Omron CX-Programmer project PampaBlanca (CX-Programmer 7.21)

# PLC PLC: CJ1M CPU13
I/O table (CPU CJ1M-CPU13): rack 0 slot 0 CJ1W-ETN21(ETN11Mode); rack 0 slot 1 CJ1W-SRM21(2CH); rack 0 slot 2 CJ1W-ID261; rack 0 slot 3 CJ1W-ID261; rack 0 slot 4 CJ1W-ID261; rack 0 slot 5 CJ1W-OD261; rack 0 slot 6 CJ1W-OD261; rack 0 slot 7 CJ1W-OD231

## Global symbols (name address type ; comment)
AFRE 2000.03 BOOL L
BLZ1 2001.06 BOOL L
BLZ2 12.02 BOOL L
BLZ4 12.03 BOOL L
BLZ5 12.04 BOOL L
BLZ6 12.05 BOOL L
EMERGENCIA W300.00 BOOL L
EVM32 2001.07 BOOL L
EVM48 2001.08 BOOL L
EVM5 2001.04 BOOL L
EVMN25 2001.05 BOOL L
EVS11 2000.04 BOOL L
EVS11_C 2000.05 BOOL L
EVS12 2000.06 BOOL L
EVS12_C 2000.07 BOOL L
EVS13P 2000.08 BOOL L
EVS13P_C 2000.09 BOOL L
EVS13S 2000.10 BOOL L
EVS13S_C 2000.11 BOOL L
HAR2 2000.00 BOOL L
HARI 2000.02 BOOL L
M1 20.00 BOOL L
M10 20.12 BOOL L
M100 19.13 BOOL L
M102 19.14 BOOL L
M103 19.15 BOOL L
M104 2002.01 BOOL L
M105 14.00 BOOL L
M106 14.01 BOOL L
M107 14.02 BOOL L
M108 14.03 BOOL L
M108A 14.04 BOOL L
M11 20.13 BOOL L
M116 14.05 BOOL L
M117 14.06 BOOL L
M117A 14.07 BOOL L
M118 14.08 BOOL L
M11A 20.14 BOOL L
M12 20.15 BOOL L
M13 21.00 BOOL L
M14 21.01 BOOL L
M15 21.02 BOOL L
M152 12.07 BOOL L
M153 14.09 BOOL L  ; BALANZA AFRECHO CONTACTOR  C93
M153Z 12.08 BOOL L
M16 21.03 BOOL L
M16A 21.04 BOOL L
M17 21.05 BOOL L
M2 20.01 BOOL L
M21 21.06 BOOL L
M22 21.07 BOOL L
M23 21.08 BOOL L
M3 20.02 BOOL L
M31 21.09 BOOL L
M32 21.10 BOOL L
M34 21.11 BOOL L
M35 21.12 BOOL L
M36 21.13 BOOL L
M37 21.14 BOOL L
M37A 21.15 BOOL L
M38 18.00 BOOL L
M3A 20.03 BOOL L
M3B 20.04 BOOL L
M4 20.05 BOOL L
M46 18.01 BOOL L
M47 18.02 BOOL L
M48 18.03 BOOL L
M5 20.06 BOOL L
M50 18.04 BOOL L
M50A 18.05 BOOL L
M51 18.06 BOOL L
M51A 18.07 BOOL L
M52 18.08 BOOL L
M53 18.09 BOOL L
M54 18.10 BOOL L
M55 18.11 BOOL L
M56 18.12 BOOL L
M58 18.13 BOOL L
M59 18.14 BOOL L
M6 20.07 BOOL L
M61 18.15 BOOL L
M62 19.00 BOOL L
M63 19.01 BOOL L
M64 19.02 BOOL L
M65 19.03 BOOL L
M69 19.04 BOOL L
M7 20.08 BOOL L
M70 19.05 BOOL L
M71 19.06 BOOL L
M73 19.07 BOOL L
M75 19.08 BOOL L
M7A 20.09 BOOL L
M8 20.10 BOOL L
M9 20.11 BOOL L
M91 2002.00 BOOL L
M95 19.09 BOOL L
M96 19.10 BOOL L
M97 19.11 BOOL L
M99 19.12 BOOL L
MI 2002.02 BOOL L
MII 2002.03 BOOL L
MN1 14.11 BOOL L
MN10 2002.06 BOOL L
MN100 2002.10 BOOL L
MN11 14.15 BOOL L
MN12 15.00 BOOL L
MN13 2002.07 BOOL L
MN14 2002.08 BOOL L
MN15 2002.09 BOOL L
MN16 15.01 BOOL L
MN17 15.02 BOOL L
MN18 15.03 BOOL L
MN2 14.12 BOOL L
MN21 15.04 BOOL L
MN24 15.05 BOOL L
MN25 15.06 BOOL L
MN26 15.07 BOOL L
MN27 15.08 BOOL L
MN28 15.09 BOOL L
MN3 14.13 BOOL L
MN35 15.12 BOOL L
MN36 15.11 BOOL L
MN37 15.10 BOOL L
MN4 14.14 BOOL L
MN9 2002.05 BOOL L
MOZD 2000.01 BOOL L
MV 2002.04 BOOL L
MVIII 14.10 BOOL L
MYFA 12.06 BOOL L
R1MN24 2001.02 BOOL L
R1MN24_C 2001.03 BOOL L
R1MN26 2001.00 BOOL L
R1MN26_C 2001.01 BOOL L
R2MN24 2002.11 BOOL L
R2MN24_C 2002.12 BOOL L
R2MN26 2000.14 BOOL L
R2MN26_C 2000.15 BOOL L
R3MN26 2000.12 BOOL L
R3MN26_C 2000.13 BOOL L
RST32 15.14 BOOL L
RST48 15.15 BOOL L
STOP W300.01 BOOL L
TBEHA 15.13 BOOL L  ; EMBOLSADO HARIN CONTACTOR C92
XBT13 2012.15 BOOL L
XEMER0 7.11 BOOL L
XEMER1 7.10 BOOL L
XFCCM32 2008.13 BOOL L
XFCCM48 2011.10 BOOL L
XFCMN24 2008.08 BOOL L
XFCMN26 2008.09 BOOL L
XFCMN37 7.04 BOOL L
XFCMVIII 2008.10 BOOL L
XFCOM32 2008.12 BOOL L
XFCOM48 2011.09 BOOL L
XHABI1 7.09 BOOL L
XM1 0.00 BOOL L
XM10 0.12 BOOL L
XM100 4.00 BOOL L
XM102 4.01 BOOL L
XM103 4.02 BOOL L
XM104 2012.14 BOOL L
XM105 4.03 BOOL L
XM106 4.04 BOOL L
XM107 4.05 BOOL L
XM108 4.06 BOOL L
XM108A 4.07 BOOL L
XM11 0.13 BOOL L
XM116 4.08 BOOL L
XM117 4.09 BOOL L
XM117A 4.10 BOOL L
XM118 4.11 BOOL L
XM11A 0.14 BOOL L
XM12 0.15 BOOL L
XM13 1.00 BOOL L
XM14 1.01 BOOL L
XM15 1.02 BOOL L
XM153 4.12 BOOL L
XM16 1.03 BOOL L
XM16A 1.04 BOOL L
XM17 1.05 BOOL L
XM2 0.01 BOOL L
XM20 1.06 BOOL L
XM21 1.07 BOOL L
XM22 1.08 BOOL L
XM23 1.09 BOOL L
XM3 0.02 BOOL L
XM31 1.10 BOOL L
XM32 1.11 BOOL L
XM34 1.12 BOOL L
XM35 1.13 BOOL L
XM36 1.14 BOOL L
XM37 1.15 BOOL L
XM37A 2.00 BOOL L
XM38 2.01 BOOL L
XM3A 0.03 BOOL L
XM3B 0.04 BOOL L
XM4 0.05 BOOL L
XM46 2.02 BOOL L
XM47 2.03 BOOL L
XM48 2.04 BOOL L
XM5 0.06 BOOL L
XM50 2.05 BOOL L
XM50A 2.06 BOOL L
XM51 2.07 BOOL L
XM51A 2.08 BOOL L
XM52 2.09 BOOL L
XM53 2.10 BOOL L
XM54 2.11 BOOL L
XM55 2.12 BOOL L
XM56 2.13 BOOL L
XM58 2.14 BOOL L
XM59 2.15 BOOL L
XM6 0.07 BOOL L
XM61 3.00 BOOL L
XM62 3.01 BOOL L
XM63 3.02 BOOL L
XM64 3.03 BOOL L
XM65 3.04 BOOL L
XM69 3.05 BOOL L
XM7 0.08 BOOL L
XM70 3.06 BOOL L
XM71 3.07 BOOL L
XM73 3.08 BOOL L
XM75 3.09 BOOL L
XM7A 0.09 BOOL L
XM8 0.10 BOOL L
XM9 0.11 BOOL L
XM91 2012.12 BOOL L
XM92 3.10 BOOL L
XM93 3.11 BOOL L
XM95 3.12 BOOL L
XM96 3.13 BOOL L
XM97 3.14 BOOL L
XM99 3.15 BOOL L
XMI 2012.05 BOOL L
XMII 2012.06 BOOL L
XMN1 4.14 BOOL L
XMN10 2012.08 BOOL L
XMN100 2012.13 BOOL L
XMN11 5.02 BOOL L
XMN12 5.03 BOOL L
XMN13 2012.09 BOOL L
XMN14 2012.10 BOOL L
XMN15 2012.11 BOOL L
XMN16 5.04 BOOL L
XMN17 5.05 BOOL L
XMN18 5.06 BOOL L
XMN2 4.15 BOOL L
XMN21 5.07 BOOL L
XMN24 5.08 BOOL L
XMN25 5.09 BOOL L
XMN26 5.10 BOOL L
XMN27 5.11 BOOL L
XMN28 5.12 BOOL L
XMN3 5.00 BOOL L
XMN35 5.13 BOOL L
XMN36 5.14 BOOL L
XMN37 5.15 BOOL L
XMN4 5.01 BOOL L
XMN9 2012.07 BOOL L
XMVIII 4.13 BOOL L
XSAS1 2011.00 BOOL L
XSAS10 2011.08 BOOL L
XSAS11 2009.00 BOOL L
XSAS12 2009.05 BOOL L
XSAS13 2009.10 BOOL L
XSAS14 2008.14 BOOL L
XSAS15 2008.15 BOOL L
XSAS2 2011.01 BOOL L
XSAS3 2011.02 BOOL L
XSAS4 2011.03 BOOL L
XSAS5 2011.04 BOOL L
XSAS6 2011.05 BOOL L
XSAS7 2008.07 BOOL L
XSAS8 2011.06 BOOL L
XSAS9 2011.07 BOOL L
XSBS11 6.07 BOOL L
XSBS12 6.08 BOOL L
XSBS13 6.09 BOOL L
XSC1M54 2010.08 BOOL L
XSC1M55 2010.10 BOOL L
XSC2M54 2010.09 BOOL L
XSC2M55 2010.11 BOOL L
XSHM5 2008.11 BOOL L
XSHMN25 2010.02 BOOL L
XSIBLZ1 2010.15 BOOL L
XSIBLZ2 6.01 BOOL L
XSIBLZ5 6.04 BOOL L
XSIBLZ6 6.06 BOOL L
XSIC1MN26 2009.14 BOOL L
XSIC1S13 2009.12 BOOL L
XSIC2MN26 2009.09 BOOL L
XSIC2S13 2010.00 BOOL L
XSIC3MN26 2009.04 BOOL L
XSICR1MN24 2010.14 BOOL L
XSICR2MN24 2012.04 BOOL L
XSICS11 2009.01 BOOL L
XSICS12 2009.07 BOOL L
XSIO1MN26 2009.13 BOOL L
XSIO1S13 2009.11 BOOL L
XSIO2MN26 2009.08 BOOL L
XSIO2S13 2009.15 BOOL L
XSIO3MN26 2009.03 BOOL L
XSIOR1MN24 2010.13 BOOL L
XSIOR2MN24 2012.03 BOOL L
XSIOS11 2009.02 BOOL L
XSIOS12 2009.06 BOOL L
XSNAMN16 7.00 BOOL L
XSNBMN16 7.01 BOOL L
XSR1M61 7.05 BOOL L
XSR2M61 7.06 BOOL L
XSRM10 6.11 BOOL L
XSRM100 6.15 BOOL L
XSRM100_A 2008.06 BOOL L
XSRM10_A 2008.02 BOOL L
XSRM11 2008.03 BOOL L
XSRM11A 6.13 BOOL L
XSRM11A_A 2008.04 BOOL L
XSRM12 6.12 BOOL L
XSRM35 7.02 BOOL L
XSRM62 2010.04 BOOL L
XSRM63 2010.05 BOOL L
XSRM64 2010.06 BOOL L
XSRM65 2010.07 BOOL L
XSRM9 6.10 BOOL L
XSRM99 6.14 BOOL L
XSRM99_A 2008.05 BOOL L
XSRM9_A 2008.01 BOOL L
XSRMN100 2012.02 BOOL L
XSRMN102 7.07 BOOL L
XSRMN103 7.08 BOOL L
XSRMN24 2010.12 BOOL L
XSRMN26 2010.03 BOOL L
XSRMN37 7.03 BOOL L
XSSBLZ1 2010.01 BOOL L
XSSBLZ2 6.00 BOOL L
XSSBLZ4 6.02 BOOL L
XSSBLZ5 6.03 BOOL L
XSSBLZ6 6.05 BOOL L
XSTMN14INF 2012.01 BOOL L
XSTMN14SUP 2012.00 BOOL L
YAFRE W499.03 BOOL L
YBLZ1 W498.06 BOOL L
YBLZ2 W506.02 BOOL L
YBLZ4 W506.03 BOOL L
YBLZ5 W506.04 BOOL L
YBLZ6 W506.05 BOOL L
YEVM32 W498.07 BOOL L
YEVM48 W498.08 BOOL L
YEVM5 W498.04 BOOL L
YEVMN25 W498.05 BOOL L
YEVS11 W499.04 BOOL L
YEVS11_C W499.05 BOOL L
YEVS12 W499.06 BOOL L
YEVS12_C W499.07 BOOL L
YEVS13P W499.08 BOOL L
YEVS13P_C W499.09 BOOL L
YEVS13S W499.10 BOOL L
YEVS13S_C W499.11 BOOL L
YHAR2 W499.00 BOOL L
YHARI W499.02 BOOL L
YM1 W500.00 BOOL L
YM10 W500.12 BOOL L
YM100 W503.13 BOOL L
YM102 W503.14 BOOL L
YM103 W503.15 BOOL L
YM104 W497.01 BOOL L
YM105 W504.00 BOOL L
YM106 W504.01 BOOL L
YM107 W504.02 BOOL L
YM108 W504.03 BOOL L
YM108A W504.04 BOOL L
YM11 W500.13 BOOL L
YM116 W504.05 BOOL L
YM117 W504.06 BOOL L
YM117A W504.07 BOOL L
YM118 W504.08 BOOL L
YM11A W500.14 BOOL L
YM12 W500.15 BOOL L
YM13 W501.00 BOOL L
YM14 W501.01 BOOL L
YM15 W501.02 BOOL L
YM152 W506.07 BOOL L
YM153 W504.09 BOOL L
YM153Z W506.08 BOOL L
YM16 W501.03 BOOL L
YM16A W501.04 BOOL L
YM17 W501.05 BOOL L
YM2 W500.01 BOOL L
YM21 W501.06 BOOL L
YM22 W501.07 BOOL L
YM23 W501.08 BOOL L
YM3 W500.02 BOOL L
YM31 W501.09 BOOL L
YM32 W501.10 BOOL L
YM34 W501.11 BOOL L
YM35 W501.12 BOOL L
YM36 W501.13 BOOL L
YM37 W501.14 BOOL L
YM37A W501.15 BOOL L
YM38 W502.00 BOOL L
YM3A W500.03 BOOL L
YM3B W500.04 BOOL L
YM4 W500.05 BOOL L
YM46 W502.01 BOOL L
YM47 W502.02 BOOL L
YM48 W502.03 BOOL L
YM5 W500.06 BOOL L
YM50 W502.04 BOOL L
YM50A W502.05 BOOL L
YM51 W502.06 BOOL L
YM51A W502.07 BOOL L
YM52 W502.08 BOOL L
YM53 W502.09 BOOL L
YM54 W502.10 BOOL L
YM55 W502.11 BOOL L
YM56 W502.12 BOOL L
YM58 W502.13 BOOL L
YM59 W502.14 BOOL L
YM6 W500.07 BOOL L
YM61 W502.15 BOOL L
YM62 W503.00 BOOL L
YM63 W503.01 BOOL L
YM64 W503.02 BOOL L
YM65 W503.03 BOOL L
YM69 W503.04 BOOL L
YM7 W500.08 BOOL L
YM70 W503.05 BOOL L
YM71 W503.06 BOOL L
YM73 W503.07 BOOL L
YM75 W503.08 BOOL L
YM7A W500.09 BOOL L
YM8 W500.10 BOOL L
YM9 W500.11 BOOL L
YM91 W497.00 BOOL L
YM95 W503.09 BOOL L
YM96 W503.10 BOOL L
YM97 W503.11 BOOL L
YM99 W503.12 BOOL L
YMI W497.02 BOOL L
YMII W497.03 BOOL L
YMN1 W504.11 BOOL L
YMN10 W497.06 BOOL L
YMN100 W497.10 BOOL L
YMN11 W504.15 BOOL L
YMN12 W505.00 BOOL L
YMN13 W497.07 BOOL L
YMN14 W497.08 BOOL L
YMN15 W497.09 BOOL L
YMN16 W505.01 BOOL L
YMN17 W505.02 BOOL L
YMN18 W505.03 BOOL L
YMN2 W504.12 BOOL L
YMN21 W505.04 BOOL L
YMN24 W505.05 BOOL L
YMN25 W505.06 BOOL L
YMN26 W505.07 BOOL L
YMN27 W505.08 BOOL L
YMN28 W505.09 BOOL L
YMN3 W504.13 BOOL L
YMN35 W505.12 BOOL L
YMN36 W505.11 BOOL L
YMN37 W505.10 BOOL L
YMN4 W504.14 BOOL L
YMN9 W497.05 BOOL L
YMOZD W499.01 BOOL L
YMV W497.04 BOOL L
YMVIII W504.10 BOOL L
YMYFA W506.06 BOOL L
YR1MN24 W498.02 BOOL L
YR1MN24_C W498.03 BOOL L
YR1MN26 W498.00 BOOL L
YR1MN26_C W498.01 BOOL L
YR2MN24 W497.11 BOOL L
YR2MN24_C W497.12 BOOL L
YR2MN26 W499.14 BOOL L
YR2MN26_C W499.15 BOOL L
YR3MN26 W499.12 BOOL L
YR3MN26_C W499.13 BOOL L
YRST32 W300.10 BOOL L
YRST48 W300.11 BOOL L
YTBEHA W505.13 BOOL L

## Program PRINCIPAL (cyclic task 0)
; MOLINO PAMPA BLANCA

### Section Emergencia

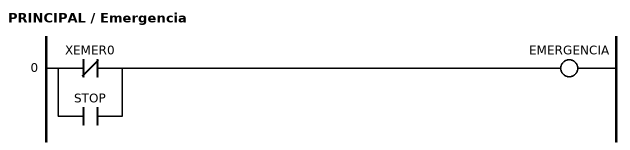
; rung 0
LDNOT XEMER0
OR STOP
OUT EMERGENCIA

### Section Llenar_Pellets_CTRL

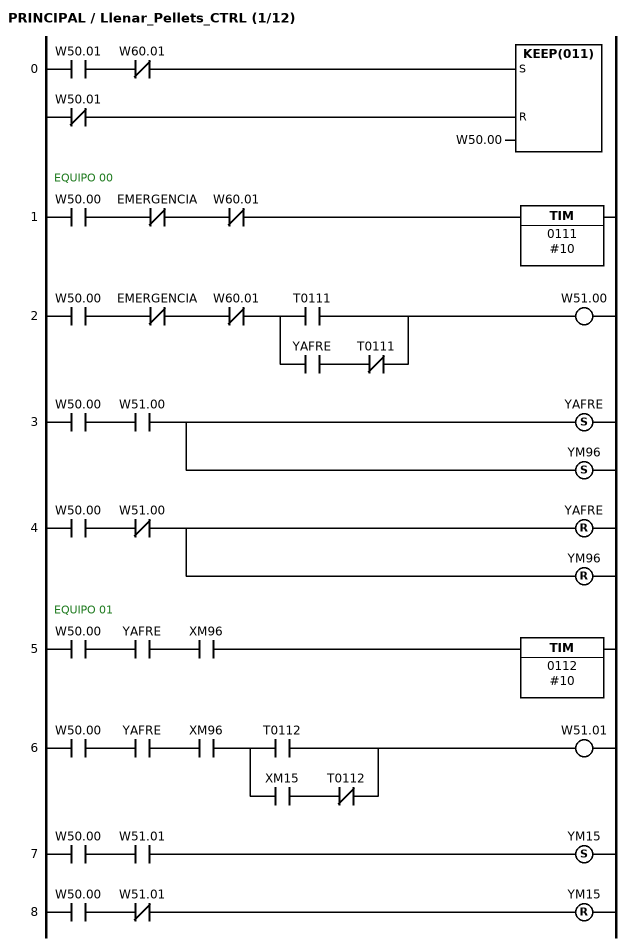
; rung 0
LD W50.01
ANDNOT W60.01
LDNOT W50.01
KEEP(011) W50.00
; rung 1: EQUIPO 00
LD W50.00
ANDNOT EMERGENCIA
ANDNOT W60.01
TIM 0111 #10
; rung 2
LD W50.00
ANDNOT EMERGENCIA
ANDNOT W60.01
LD T0111
LD YAFRE
ANDNOT T0111
ORLD
ANDLD
OUT W51.00
; rung 3
LD W50.00
AND W51.00
SET YAFRE
SET YM96
; rung 4
LD W50.00
ANDNOT W51.00
RSET YAFRE
RSET YM96
; rung 5: EQUIPO 01
LD W50.00
AND YAFRE
AND XM96
TIM 0112 #10
; rung 6
LD W50.00
AND YAFRE
AND XM96
LD T0112
LD XM15
ANDNOT T0112
ORLD
ANDLD
OUT W51.01
; rung 7
LD W50.00
AND W51.01
SET YM15
; rung 8
LD W50.00
ANDNOT W51.01
RSET YM15

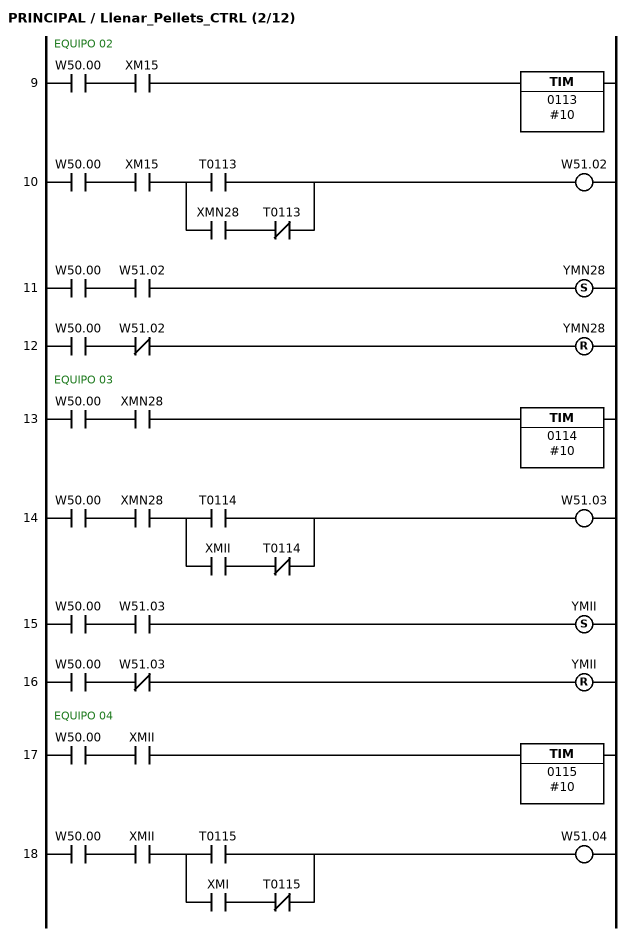
; rung 9: EQUIPO 02
LD W50.00
AND XM15
TIM 0113 #10
; rung 10
LD W50.00
AND XM15
LD T0113
LD XMN28
ANDNOT T0113
ORLD
ANDLD
OUT W51.02
; rung 11
LD W50.00
AND W51.02
SET YMN28
; rung 12
LD W50.00
ANDNOT W51.02
RSET YMN28
; rung 13: EQUIPO 03
LD W50.00
AND XMN28
TIM 0114 #10
; rung 14
LD W50.00
AND XMN28
LD T0114
LD XMII
ANDNOT T0114
ORLD
ANDLD
OUT W51.03
; rung 15
LD W50.00
AND W51.03
SET YMII
; rung 16
LD W50.00
ANDNOT W51.03
RSET YMII
; rung 17: EQUIPO 04
LD W50.00
AND XMII
TIM 0115 #10
; rung 18
LD W50.00
AND XMII
LD T0115
LD XMI
ANDNOT T0115
ORLD
ANDLD
OUT W51.04

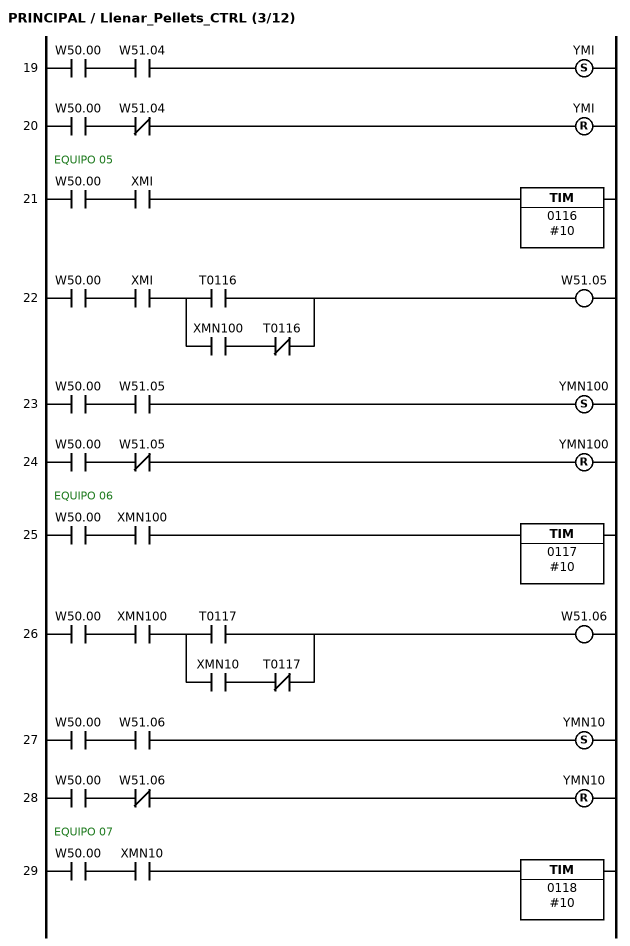
; rung 19
LD W50.00
AND W51.04
SET YMI
; rung 20
LD W50.00
ANDNOT W51.04
RSET YMI
; rung 21: EQUIPO 05
LD W50.00
AND XMI
TIM 0116 #10
; rung 22
LD W50.00
AND XMI
LD T0116
LD XMN100
ANDNOT T0116
ORLD
ANDLD
OUT W51.05
; rung 23
LD W50.00
AND W51.05
SET YMN100
; rung 24
LD W50.00
ANDNOT W51.05
RSET YMN100
; rung 25: EQUIPO 06
LD W50.00
AND XMN100
TIM 0117 #10
; rung 26
LD W50.00
AND XMN100
LD T0117
LD XMN10
ANDNOT T0117
ORLD
ANDLD
OUT W51.06
; rung 27
LD W50.00
AND W51.06
SET YMN10
; rung 28
LD W50.00
ANDNOT W51.06
RSET YMN10
; rung 29: EQUIPO 07
LD W50.00
AND XMN10
TIM 0118 #10

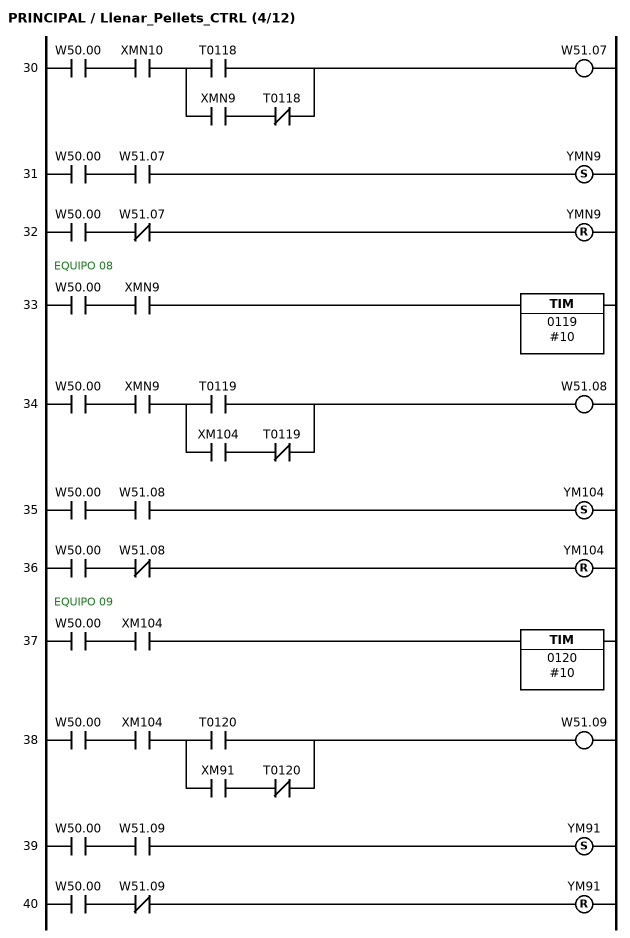
; rung 30
LD W50.00
AND XMN10
LD T0118
LD XMN9
ANDNOT T0118
ORLD
ANDLD
OUT W51.07
; rung 31
LD W50.00
AND W51.07
SET YMN9
; rung 32
LD W50.00
ANDNOT W51.07
RSET YMN9
; rung 33: EQUIPO 08
LD W50.00
AND XMN9
TIM 0119 #10
; rung 34
LD W50.00
AND XMN9
LD T0119
LD XM104
ANDNOT T0119
ORLD
ANDLD
OUT W51.08
; rung 35
LD W50.00
AND W51.08
SET YM104
; rung 36
LD W50.00
ANDNOT W51.08
RSET YM104
; rung 37: EQUIPO 09
LD W50.00
AND XM104
TIM 0120 #10
; rung 38
LD W50.00
AND XM104
LD T0120
LD XM91
ANDNOT T0120
ORLD
ANDLD
OUT W51.09
; rung 39
LD W50.00
AND W51.09
SET YM91
; rung 40
LD W50.00
ANDNOT W51.09
RSET YM91

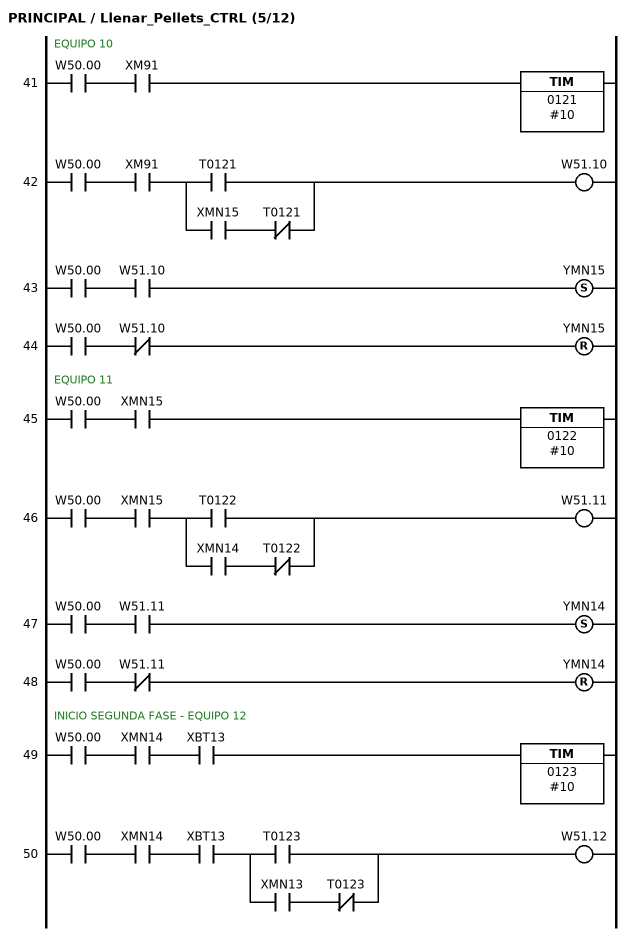
; rung 41: EQUIPO 10
LD W50.00
AND XM91
TIM 0121 #10
; rung 42
LD W50.00
AND XM91
LD T0121
LD XMN15
ANDNOT T0121
ORLD
ANDLD
OUT W51.10
; rung 43
LD W50.00
AND W51.10
SET YMN15
; rung 44
LD W50.00
ANDNOT W51.10
RSET YMN15
; rung 45: EQUIPO 11
LD W50.00
AND XMN15
TIM 0122 #10
; rung 46
LD W50.00
AND XMN15
LD T0122
LD XMN14
ANDNOT T0122
ORLD
ANDLD
OUT W51.11
; rung 47
LD W50.00
AND W51.11
SET YMN14
; rung 48
LD W50.00
ANDNOT W51.11
RSET YMN14
; rung 49: INICIO SEGUNDA FASE - EQUIPO 12
LD W50.00
AND XMN14
AND XBT13
TIM 0123 #10
; rung 50
LD W50.00
AND XMN14
AND XBT13
LD T0123
LD XMN13
ANDNOT T0123
ORLD
ANDLD
OUT W51.12

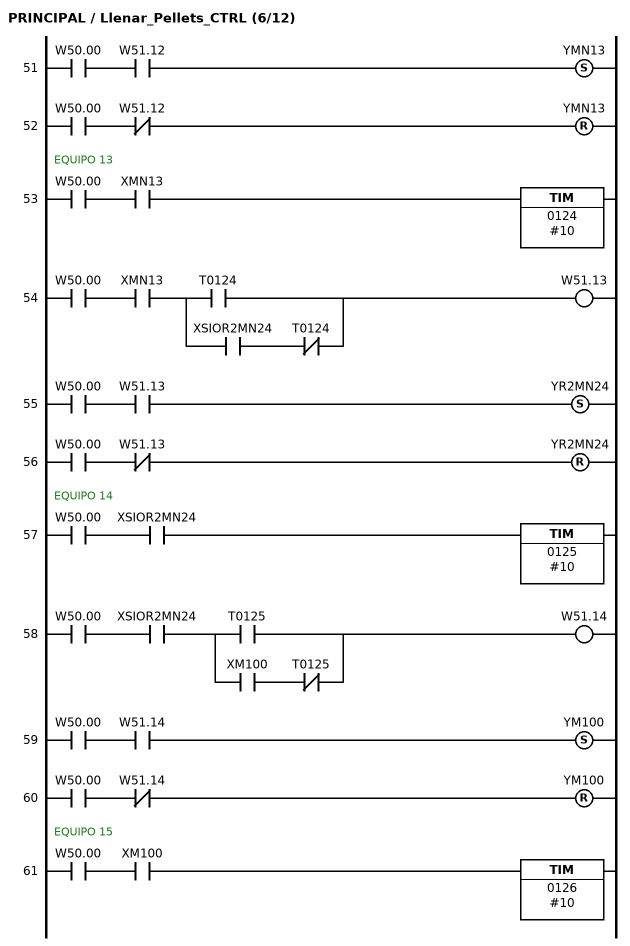
; rung 51
LD W50.00
AND W51.12
SET YMN13
; rung 52
LD W50.00
ANDNOT W51.12
RSET YMN13
; rung 53: EQUIPO 13
LD W50.00
AND XMN13
TIM 0124 #10
; rung 54
LD W50.00
AND XMN13
LD T0124
LD XSIOR2MN24
ANDNOT T0124
ORLD
ANDLD
OUT W51.13
; rung 55
LD W50.00
AND W51.13
SET YR2MN24
; rung 56
LD W50.00
ANDNOT W51.13
RSET YR2MN24
; rung 57: EQUIPO 14
LD W50.00
AND XSIOR2MN24
TIM 0125 #10
; rung 58
LD W50.00
AND XSIOR2MN24
LD T0125
LD XM100
ANDNOT T0125
ORLD
ANDLD
OUT W51.14
; rung 59
LD W50.00
AND W51.14
SET YM100
; rung 60
LD W50.00
ANDNOT W51.14
RSET YM100
; rung 61: EQUIPO 15
LD W50.00
AND XM100
TIM 0126 #10

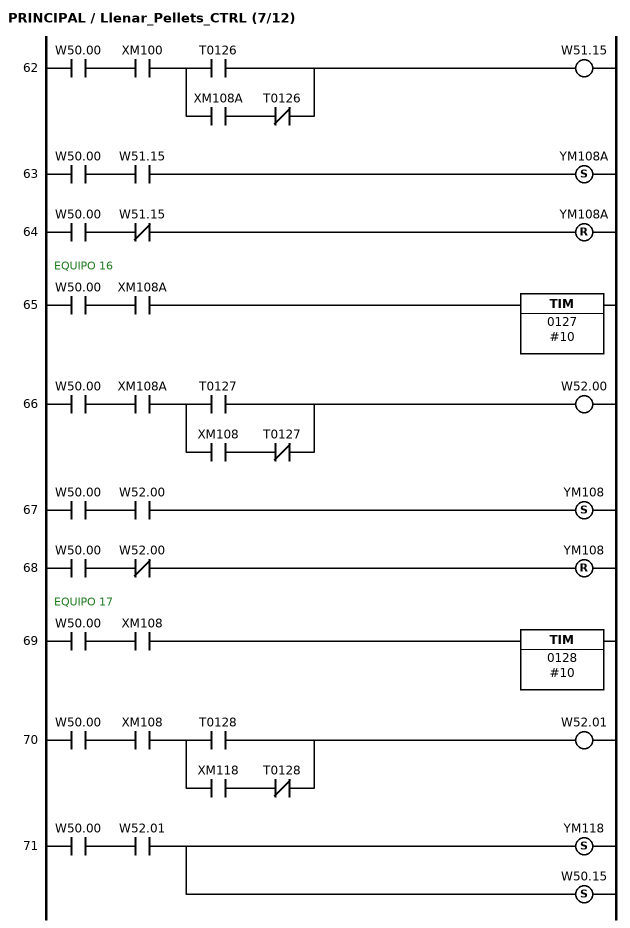
; rung 62
LD W50.00
AND XM100
LD T0126
LD XM108A
ANDNOT T0126
ORLD
ANDLD
OUT W51.15
; rung 63
LD W50.00
AND W51.15
SET YM108A
; rung 64
LD W50.00
ANDNOT W51.15
RSET YM108A
; rung 65: EQUIPO 16
LD W50.00
AND XM108A
TIM 0127 #10
; rung 66
LD W50.00
AND XM108A
LD T0127
LD XM108
ANDNOT T0127
ORLD
ANDLD
OUT W52.00
; rung 67
LD W50.00
AND W52.00
SET YM108
; rung 68
LD W50.00
ANDNOT W52.00
RSET YM108
; rung 69: EQUIPO 17
LD W50.00
AND XM108
TIM 0128 #10
; rung 70
LD W50.00
AND XM108
LD T0128
LD XM118
ANDNOT T0128
ORLD
ANDLD
OUT W52.01
; rung 71
LD W50.00
AND W52.01
SET YM118
SET W50.15

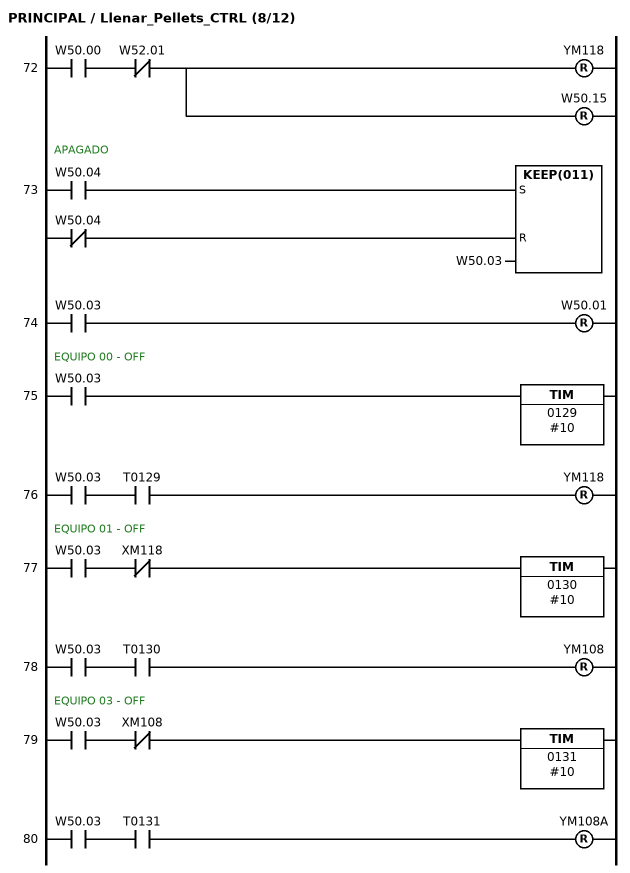
; rung 72
LD W50.00
ANDNOT W52.01
RSET YM118
RSET W50.15
; rung 73: APAGADO
LD W50.04
LDNOT W50.04
KEEP(011) W50.03
; rung 74
LD W50.03
RSET W50.01
; rung 75: EQUIPO 00 - OFF
LD W50.03
TIM 0129 #10
; rung 76
LD W50.03
AND T0129
RSET YM118
; rung 77: EQUIPO 01 - OFF
LD W50.03
ANDNOT XM118
TIM 0130 #10
; rung 78
LD W50.03
AND T0130
RSET YM108
; rung 79: EQUIPO 03 - OFF
LD W50.03
ANDNOT XM108
TIM 0131 #10
; rung 80
LD W50.03
AND T0131
RSET YM108A

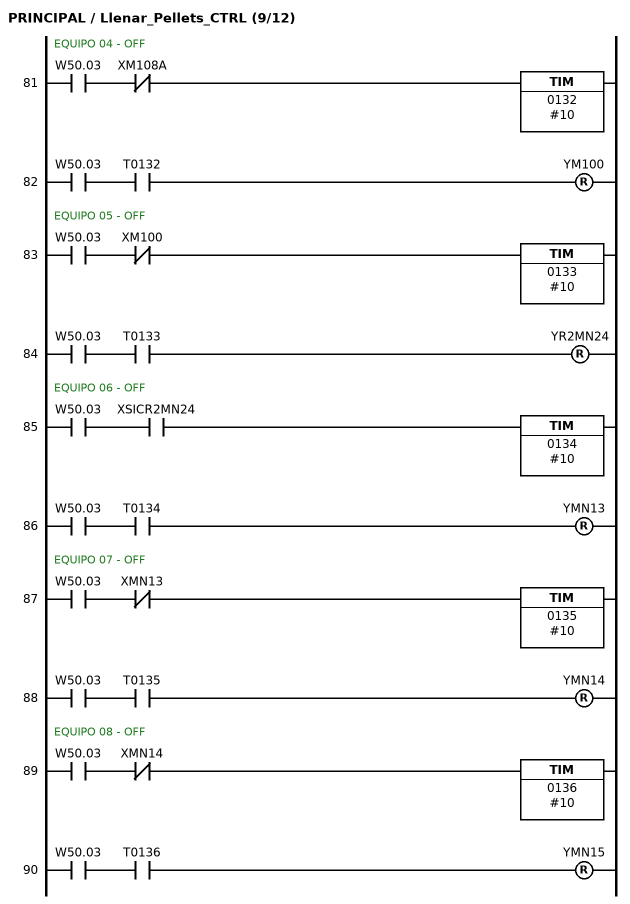
; rung 81: EQUIPO 04 - OFF
LD W50.03
ANDNOT XM108A
TIM 0132 #10
; rung 82
LD W50.03
AND T0132
RSET YM100
; rung 83: EQUIPO 05 - OFF
LD W50.03
ANDNOT XM100
TIM 0133 #10
; rung 84
LD W50.03
AND T0133
RSET YR2MN24
; rung 85: EQUIPO 06 - OFF
LD W50.03
AND XSICR2MN24
TIM 0134 #10
; rung 86
LD W50.03
AND T0134
RSET YMN13
; rung 87: EQUIPO 07 - OFF
LD W50.03
ANDNOT XMN13
TIM 0135 #10
; rung 88
LD W50.03
AND T0135
RSET YMN14
; rung 89: EQUIPO 08 - OFF
LD W50.03
ANDNOT XMN14
TIM 0136 #10
; rung 90
LD W50.03
AND T0136
RSET YMN15

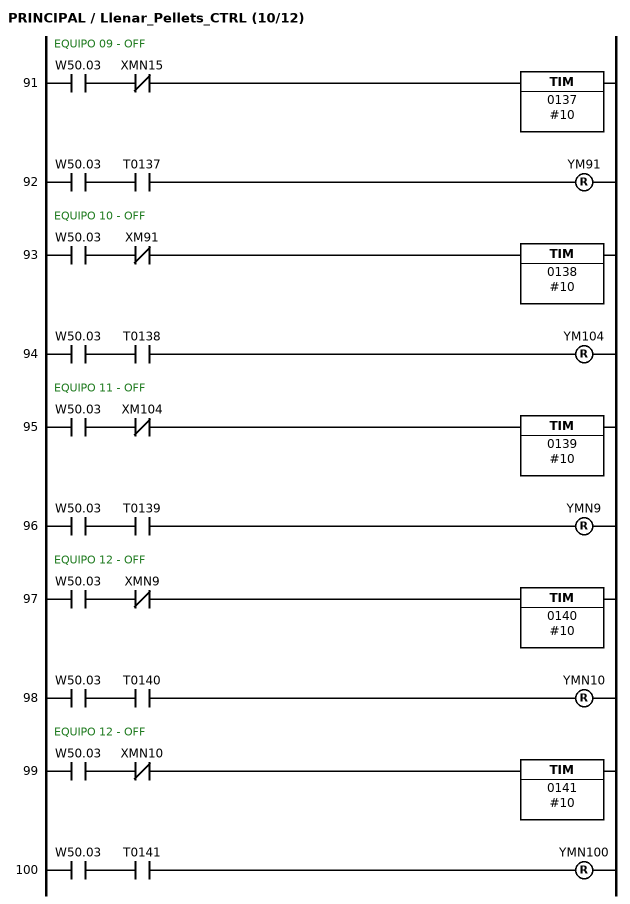
; rung 91: EQUIPO 09 - OFF
LD W50.03
ANDNOT XMN15
TIM 0137 #10
; rung 92
LD W50.03
AND T0137
RSET YM91
; rung 93: EQUIPO 10 - OFF
LD W50.03
ANDNOT XM91
TIM 0138 #10
; rung 94
LD W50.03
AND T0138
RSET YM104
; rung 95: EQUIPO 11 - OFF
LD W50.03
ANDNOT XM104
TIM 0139 #10
; rung 96
LD W50.03
AND T0139
RSET YMN9
; rung 97: EQUIPO 12 - OFF
LD W50.03
ANDNOT XMN9
TIM 0140 #10
; rung 98
LD W50.03
AND T0140
RSET YMN10
; rung 99: EQUIPO 12 - OFF
LD W50.03
ANDNOT XMN10
TIM 0141 #10
; rung 100
LD W50.03
AND T0141
RSET YMN100

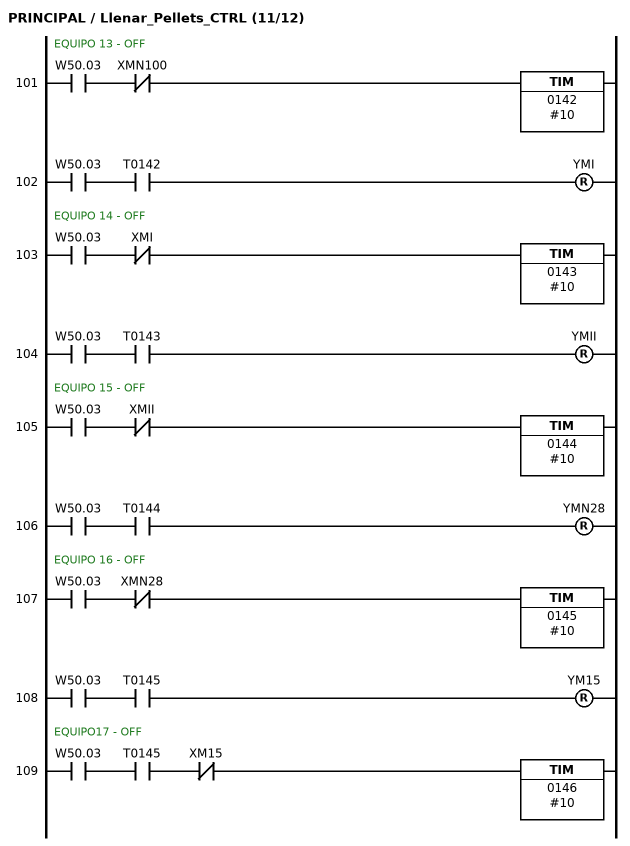
; rung 101: EQUIPO 13 - OFF
LD W50.03
ANDNOT XMN100
TIM 0142 #10
; rung 102
LD W50.03
AND T0142
RSET YMI
; rung 103: EQUIPO 14 - OFF
LD W50.03
ANDNOT XMI
TIM 0143 #10
; rung 104
LD W50.03
AND T0143
RSET YMII
; rung 105: EQUIPO 15 - OFF
LD W50.03
ANDNOT XMII
TIM 0144 #10
; rung 106
LD W50.03
AND T0144
RSET YMN28
; rung 107: EQUIPO 16 - OFF
LD W50.03
ANDNOT XMN28
TIM 0145 #10
; rung 108
LD W50.03
AND T0145
RSET YM15
; rung 109: EQUIPO17 - OFF
LD W50.03
AND T0145
ANDNOT XM15
TIM 0146 #10

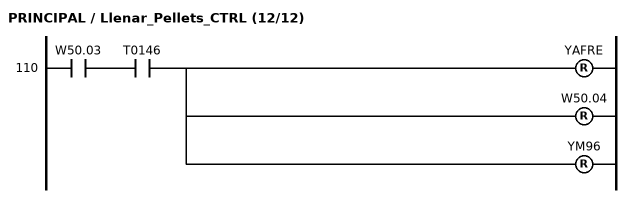
; rung 110
LD W50.03
AND T0146
RSET YAFRE
RSET W50.04
RSET YM96

### Section Llenar_Afrecho_CTRL

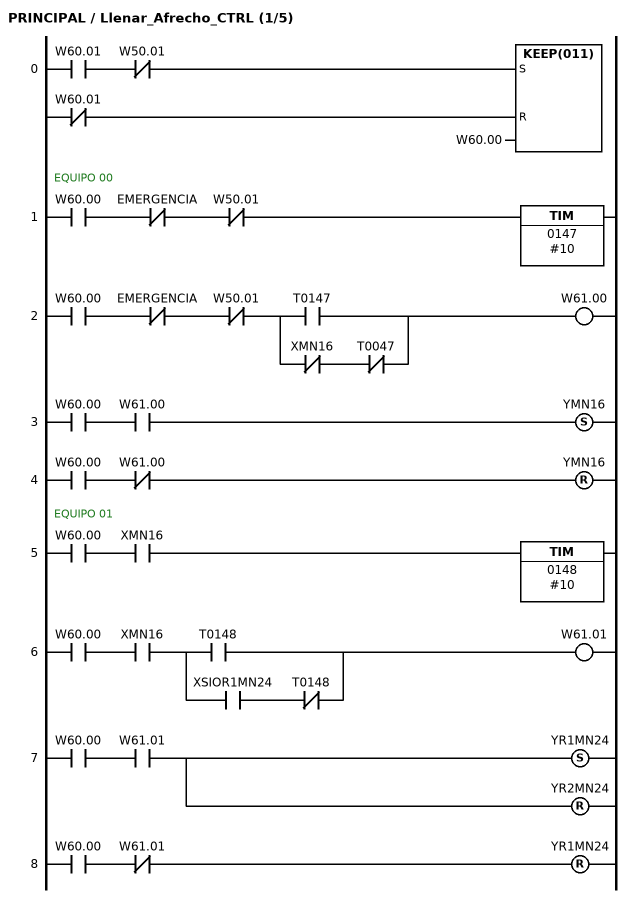
; rung 0
LD W60.01
ANDNOT W50.01
LDNOT W60.01
KEEP(011) W60.00
; rung 1: EQUIPO 00
LD W60.00
ANDNOT EMERGENCIA
ANDNOT W50.01
TIM 0147 #10
; rung 2
LD W60.00
ANDNOT EMERGENCIA
ANDNOT W50.01
LD T0147
LDNOT XMN16
ANDNOT T0047
ORLD
ANDLD
OUT W61.00
; rung 3
LD W60.00
AND W61.00
SET YMN16
; rung 4
LD W60.00
ANDNOT W61.00
RSET YMN16
; rung 5: EQUIPO 01
LD W60.00
AND XMN16
TIM 0148 #10
; rung 6
LD W60.00
AND XMN16
LD T0148
LD XSIOR1MN24
ANDNOT T0148
ORLD
ANDLD
OUT W61.01
; rung 7
LD W60.00
AND W61.01
SET YR1MN24
RSET YR2MN24
; rung 8
LD W60.00
ANDNOT W61.01
RSET YR1MN24

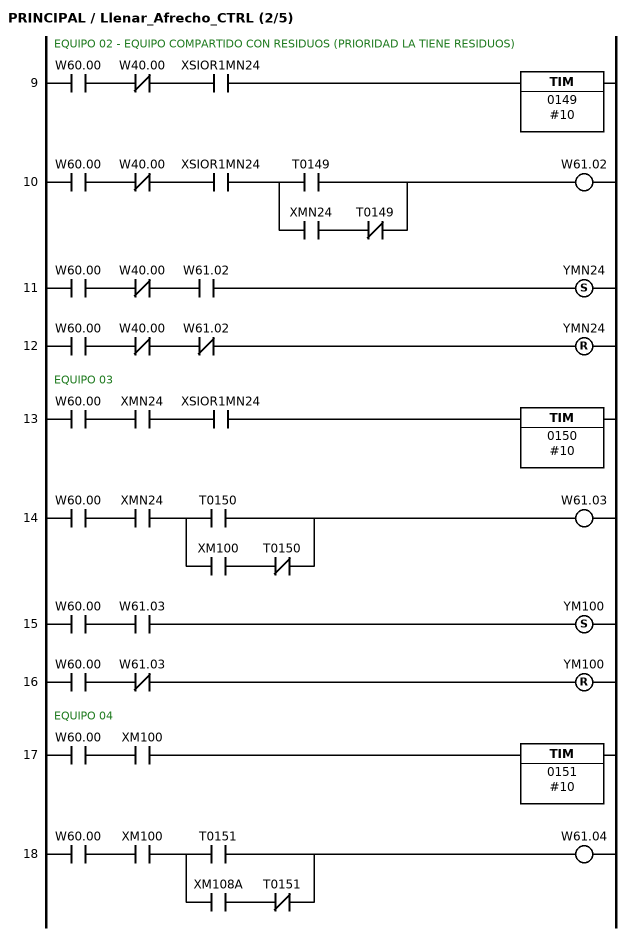
; rung 9: EQUIPO 02 - EQUIPO COMPARTIDO CON RESIDUOS (PRIORIDAD LA TIENE RESIDUOS)
LD W60.00
ANDNOT W40.00
AND XSIOR1MN24
TIM 0149 #10
; rung 10
LD W60.00
ANDNOT W40.00
AND XSIOR1MN24
LD T0149
LD XMN24
ANDNOT T0149
ORLD
ANDLD
OUT W61.02
; rung 11
LD W60.00
ANDNOT W40.00
AND W61.02
SET YMN24
; rung 12
LD W60.00
ANDNOT W40.00
ANDNOT W61.02
RSET YMN24
; rung 13: EQUIPO 03
LD W60.00
AND XMN24
AND XSIOR1MN24
TIM 0150 #10
; rung 14
LD W60.00
AND XMN24
LD T0150
LD XM100
ANDNOT T0150
ORLD
ANDLD
OUT W61.03
; rung 15
LD W60.00
AND W61.03
SET YM100
; rung 16
LD W60.00
ANDNOT W61.03
RSET YM100
; rung 17: EQUIPO 04
LD W60.00
AND XM100
TIM 0151 #10
; rung 18
LD W60.00
AND XM100
LD T0151
LD XM108A
ANDNOT T0151
ORLD
ANDLD
OUT W61.04

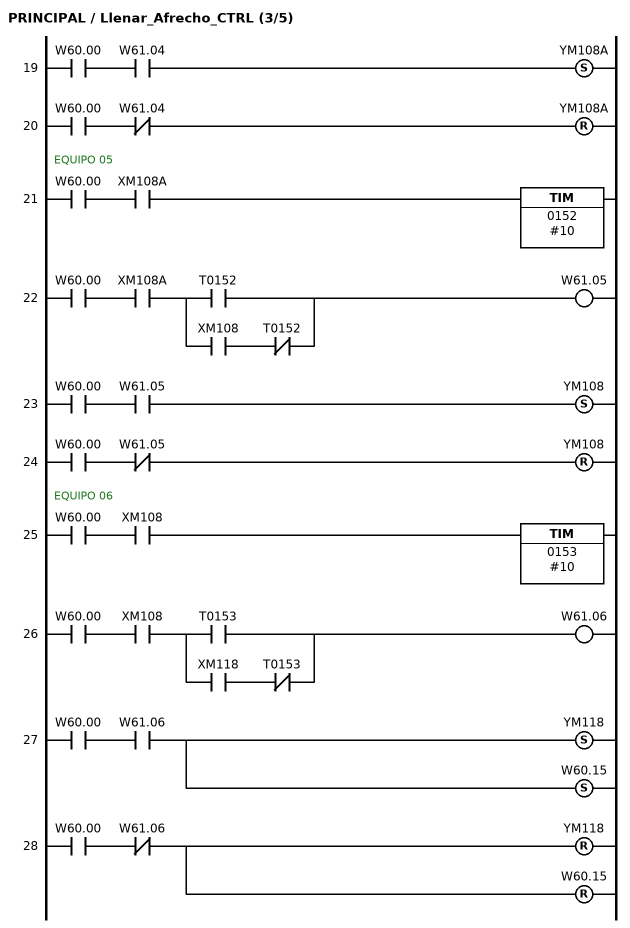
; rung 19
LD W60.00
AND W61.04
SET YM108A
; rung 20
LD W60.00
ANDNOT W61.04
RSET YM108A
; rung 21: EQUIPO 05
LD W60.00
AND XM108A
TIM 0152 #10
; rung 22
LD W60.00
AND XM108A
LD T0152
LD XM108
ANDNOT T0152
ORLD
ANDLD
OUT W61.05
; rung 23
LD W60.00
AND W61.05
SET YM108
; rung 24
LD W60.00
ANDNOT W61.05
RSET YM108
; rung 25: EQUIPO 06
LD W60.00
AND XM108
TIM 0153 #10
; rung 26
LD W60.00
AND XM108
LD T0153
LD XM118
ANDNOT T0153
ORLD
ANDLD
OUT W61.06
; rung 27
LD W60.00
AND W61.06
SET YM118
SET W60.15
; rung 28
LD W60.00
ANDNOT W61.06
RSET YM118
RSET W60.15

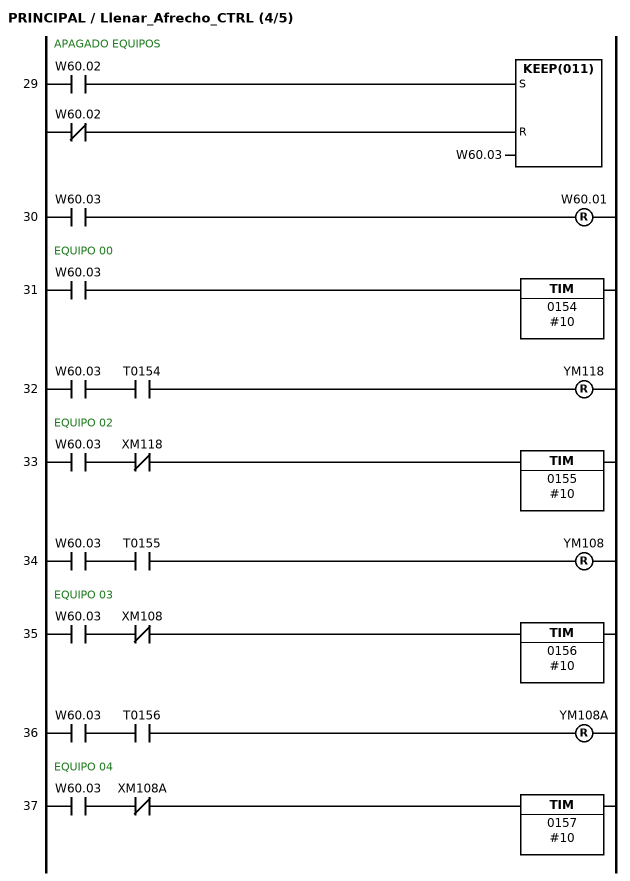
; rung 29: APAGADO EQUIPOS
LD W60.02
LDNOT W60.02
KEEP(011) W60.03
; rung 30
LD W60.03
RSET W60.01
; rung 31: EQUIPO 00
LD W60.03
TIM 0154 #10
; rung 32
LD W60.03
AND T0154
RSET YM118
; rung 33: EQUIPO 02
LD W60.03
ANDNOT XM118
TIM 0155 #10
; rung 34
LD W60.03
AND T0155
RSET YM108
; rung 35: EQUIPO 03
LD W60.03
ANDNOT XM108
TIM 0156 #10
; rung 36
LD W60.03
AND T0156
RSET YM108A
; rung 37: EQUIPO 04
LD W60.03
ANDNOT XM108A
TIM 0157 #10

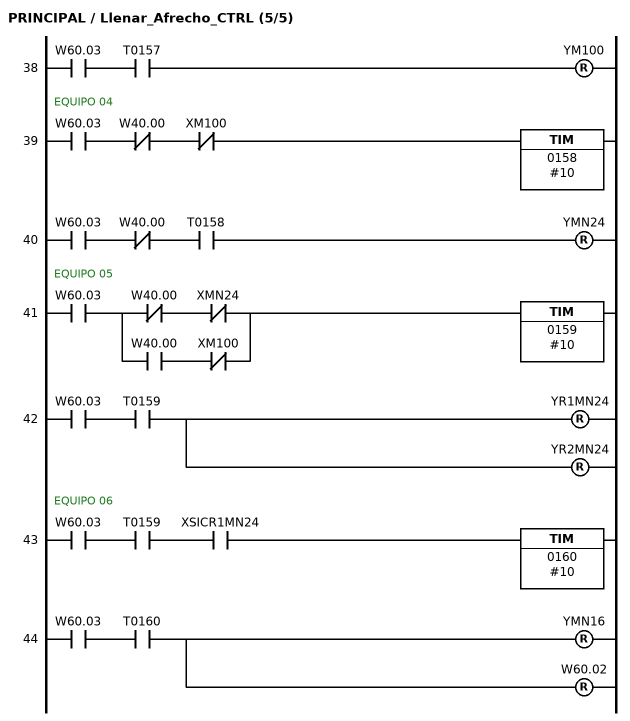
; rung 38
LD W60.03
AND T0157
RSET YM100
; rung 39: EQUIPO 04
LD W60.03
ANDNOT W40.00
ANDNOT XM100
TIM 0158 #10
; rung 40
LD W60.03
ANDNOT W40.00
AND T0158
RSET YMN24
; rung 41: EQUIPO 05
LD W60.03
LDNOT W40.00
ANDNOT XMN24
LD W40.00
ANDNOT XM100
ORLD
ANDLD
TIM 0159 #10
; rung 42
LD W60.03
AND T0159
RSET YR1MN24
RSET YR2MN24
; rung 43: EQUIPO 06
LD W60.03
AND T0159
AND XSICR1MN24
TIM 0160 #10
; rung 44
LD W60.03
AND T0160
RSET YMN16
RSET W60.02

### Section Afrecho_Pellets_OUT

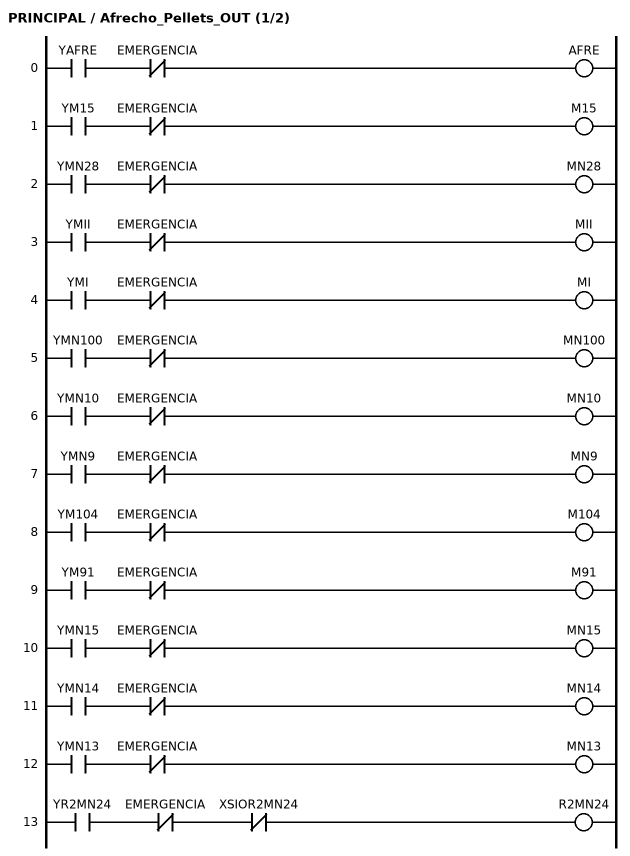
; rung 0
LD YAFRE
ANDNOT EMERGENCIA
OUT AFRE
; rung 1
LD YM15
ANDNOT EMERGENCIA
OUT M15
; rung 2
LD YMN28
ANDNOT EMERGENCIA
OUT MN28
; rung 3
LD YMII
ANDNOT EMERGENCIA
OUT MII
; rung 4
LD YMI
ANDNOT EMERGENCIA
OUT MI
; rung 5
LD YMN100
ANDNOT EMERGENCIA
OUT MN100
; rung 6
LD YMN10
ANDNOT EMERGENCIA
OUT MN10
; rung 7
LD YMN9
ANDNOT EMERGENCIA
OUT MN9
; rung 8
LD YM104
ANDNOT EMERGENCIA
OUT M104
; rung 9
LD YM91
ANDNOT EMERGENCIA
OUT M91
; rung 10
LD YMN15
ANDNOT EMERGENCIA
OUT MN15
; rung 11
LD YMN14
ANDNOT EMERGENCIA
OUT MN14
; rung 12
LD YMN13
ANDNOT EMERGENCIA
OUT MN13
; rung 13
LD YR2MN24
ANDNOT EMERGENCIA
ANDNOT XSIOR2MN24
OUT R2MN24

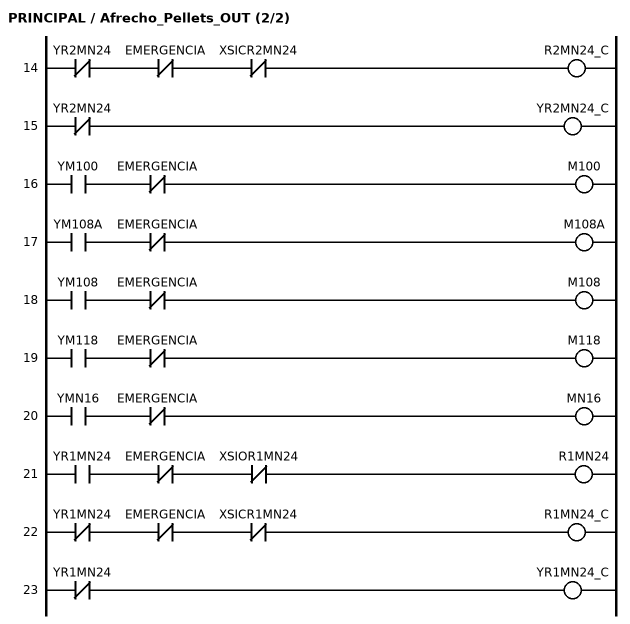
; rung 14
LDNOT YR2MN24
ANDNOT EMERGENCIA
ANDNOT XSICR2MN24
OUT R2MN24_C
; rung 15
LDNOT YR2MN24
OUT YR2MN24_C
; rung 16
LD YM100
ANDNOT EMERGENCIA
OUT M100
; rung 17
LD YM108A
ANDNOT EMERGENCIA
OUT M108A
; rung 18
LD YM108
ANDNOT EMERGENCIA
OUT M108
; rung 19
LD YM118
ANDNOT EMERGENCIA
OUT M118
; rung 20
LD YMN16
ANDNOT EMERGENCIA
OUT MN16
; rung 21
LD YR1MN24
ANDNOT EMERGENCIA
ANDNOT XSIOR1MN24
OUT R1MN24
; rung 22
LDNOT YR1MN24
ANDNOT EMERGENCIA
ANDNOT XSICR1MN24
OUT R1MN24_C
; rung 23
LDNOT YR1MN24
OUT YR1MN24_C

### Section Terminados_CTRL

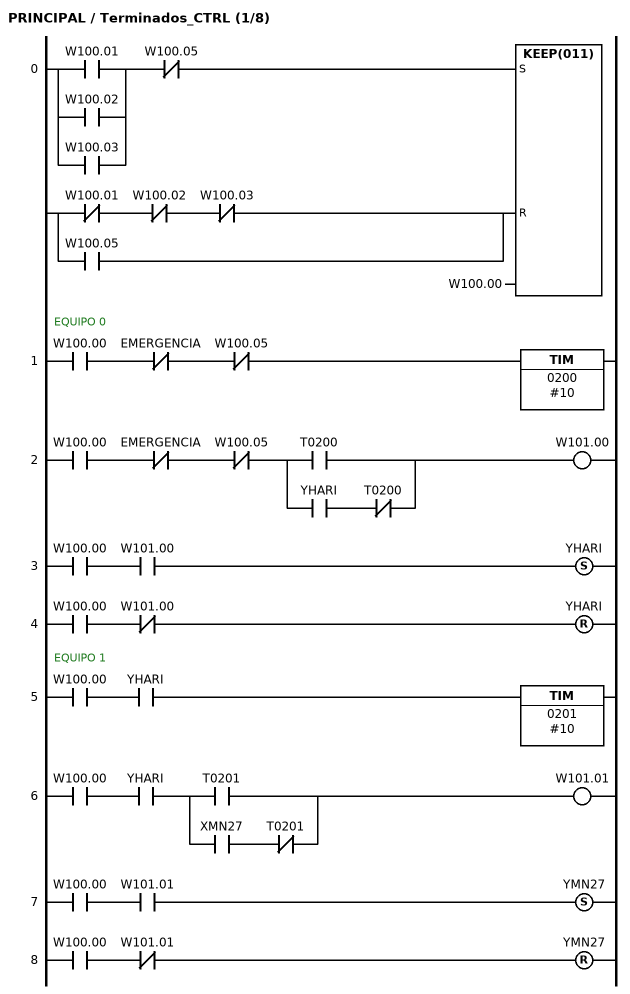
; rung 0
LD W100.01
OR W100.02
OR W100.03
ANDNOT W100.05
LDNOT W100.01
ANDNOT W100.02
ANDNOT W100.03
OR W100.05
KEEP(011) W100.00
; rung 1: EQUIPO 0
LD W100.00
ANDNOT EMERGENCIA
ANDNOT W100.05
TIM 0200 #10
; rung 2
LD W100.00
ANDNOT EMERGENCIA
ANDNOT W100.05
LD T0200
LD YHARI
ANDNOT T0200
ORLD
ANDLD
OUT W101.00
; rung 3
LD W100.00
AND W101.00
SET YHARI
; rung 4
LD W100.00
ANDNOT W101.00
RSET YHARI
; rung 5: EQUIPO 1
LD W100.00
AND YHARI
TIM 0201 #10
; rung 6
LD W100.00
AND YHARI
LD T0201
LD XMN27
ANDNOT T0201
ORLD
ANDLD
OUT W101.01
; rung 7
LD W100.00
AND W101.01
SET YMN27
; rung 8
LD W100.00
ANDNOT W101.01
RSET YMN27

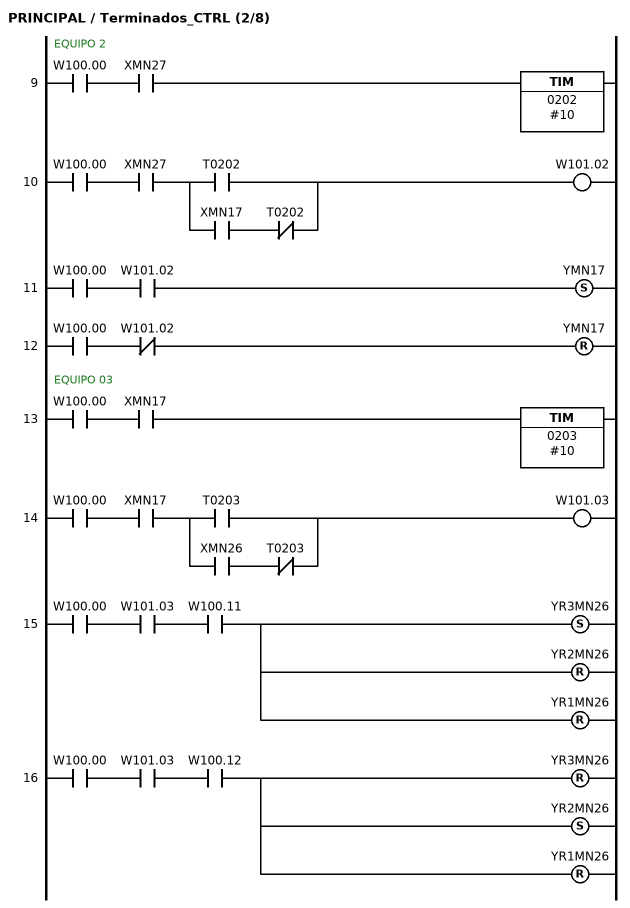
; rung 9: EQUIPO 2
LD W100.00
AND XMN27
TIM 0202 #10
; rung 10
LD W100.00
AND XMN27
LD T0202
LD XMN17
ANDNOT T0202
ORLD
ANDLD
OUT W101.02
; rung 11
LD W100.00
AND W101.02
SET YMN17
; rung 12
LD W100.00
ANDNOT W101.02
RSET YMN17
; rung 13: EQUIPO 03
LD W100.00
AND XMN17
TIM 0203 #10
; rung 14
LD W100.00
AND XMN17
LD T0203
LD XMN26
ANDNOT T0203
ORLD
ANDLD
OUT W101.03
; rung 15
LD W100.00
AND W101.03
AND W100.11
SET YR3MN26
RSET YR2MN26
RSET YR1MN26
; rung 16
LD W100.00
AND W101.03
AND W100.12
RSET YR3MN26
SET YR2MN26
RSET YR1MN26

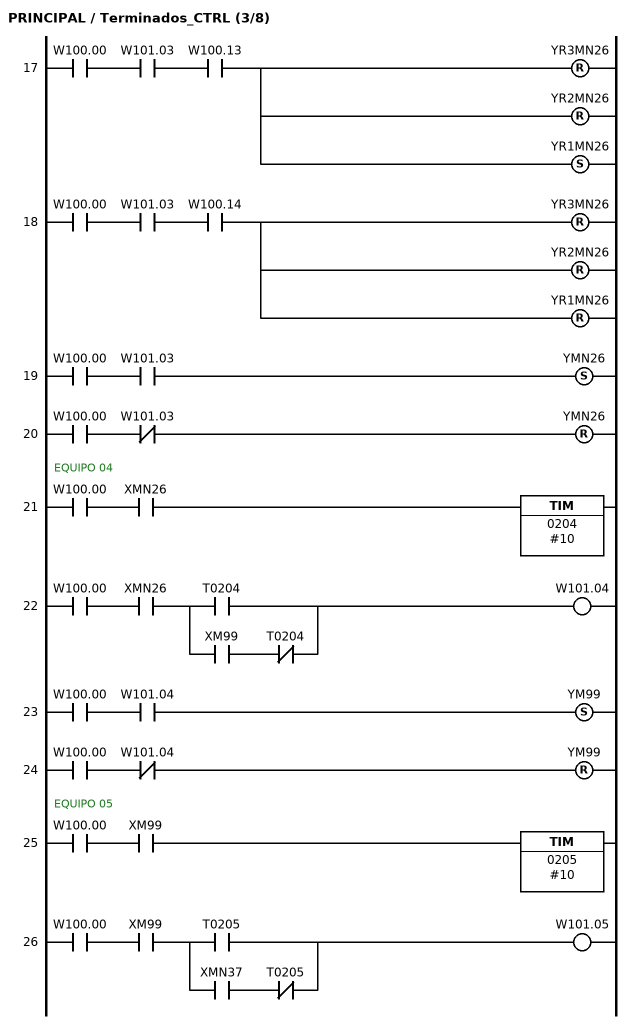
; rung 17
LD W100.00
AND W101.03
AND W100.13
RSET YR3MN26
RSET YR2MN26
SET YR1MN26
; rung 18
LD W100.00
AND W101.03
AND W100.14
RSET YR3MN26
RSET YR2MN26
RSET YR1MN26
; rung 19
LD W100.00
AND W101.03
SET YMN26
; rung 20
LD W100.00
ANDNOT W101.03
RSET YMN26
; rung 21: EQUIPO 04
LD W100.00
AND XMN26
TIM 0204 #10
; rung 22
LD W100.00
AND XMN26
LD T0204
LD XM99
ANDNOT T0204
ORLD
ANDLD
OUT W101.04
; rung 23
LD W100.00
AND W101.04
SET YM99
; rung 24
LD W100.00
ANDNOT W101.04
RSET YM99
; rung 25: EQUIPO 05
LD W100.00
AND XM99
TIM 0205 #10
; rung 26
LD W100.00
AND XM99
LD T0205
LD XMN37
ANDNOT T0205
ORLD
ANDLD
OUT W101.05

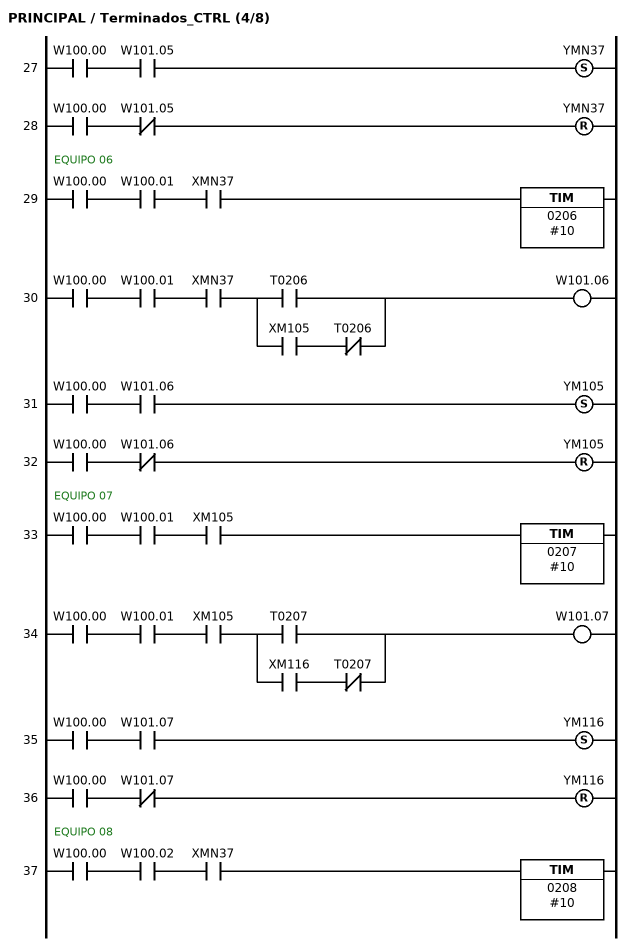
; rung 27
LD W100.00
AND W101.05
SET YMN37
; rung 28
LD W100.00
ANDNOT W101.05
RSET YMN37
; rung 29: EQUIPO 06
LD W100.00
AND W100.01
AND XMN37
TIM 0206 #10
; rung 30
LD W100.00
AND W100.01
AND XMN37
LD T0206
LD XM105
ANDNOT T0206
ORLD
ANDLD
OUT W101.06
; rung 31
LD W100.00
AND W101.06
SET YM105
; rung 32
LD W100.00
ANDNOT W101.06
RSET YM105
; rung 33: EQUIPO 07
LD W100.00
AND W100.01
AND XM105
TIM 0207 #10
; rung 34
LD W100.00
AND W100.01
AND XM105
LD T0207
LD XM116
ANDNOT T0207
ORLD
ANDLD
OUT W101.07
; rung 35
LD W100.00
AND W101.07
SET YM116
; rung 36
LD W100.00
ANDNOT W101.07
RSET YM116
; rung 37: EQUIPO 08
LD W100.00
AND W100.02
AND XMN37
TIM 0208 #10

